FUNCTION_BLOCK AxisHalt IMPLEMENTS I_Task
VAR_INPUT
END_VAR
VAR_OUTPUT
END_VAR
VAR
	mcHalt : Tc2_MC2.MC_Halt;
	_Axis : REFERENCE TO Tc2_MC2.AXIS_REF;
	_Halt : BOOL;
	State: INT;
	_Done: BOOL;
	_Error: BOOL;
	_Busy: BOOL;
END_VAR

{analysis -2}

METHOD Abort : BOOL
mcHalt.Execute := FALSE;
_Busy := FALSE;
_Halt := FALSE;
Abort := TRUE;
State := 0;
END_METHOD

PROPERTY Busy : BOOL
GET
Busy := _Busy;
END_GET
END_PROPERTY

METHOD Cycle : HRESULT
VAR_INPUT
END_VAR
Cycle := S_OK;
CASE State OF
	0:
		IF _Halt THEN
			Cycle := S_PENDING;
			_Done := FALSE;
			_Error := FALSE;
			_Busy := TRUE;
			mcHalt.Execute := TRUE;
			IF mcHalt.Busy THEN
				State := 10;
				_Halt := FALSE;
			END_IF
		END_IF
	
	10:
		IF NOT mcHalt.Busy THEN
			IF mcHalt.Done THEN
				_Done := TRUE;
			ELSIF mcHalt.Error THEN
				_Error := TRUE;
			END_IF
			_Busy := FALSE;
			mcHalt.Execute := FALSE;
			State := 0;
			Cycle := S_OK;
		END_IF
	ELSE
		Cycle := E_FAIL;
END_CASE

mcHalt(Axis := _Axis);
END_METHOD

PROPERTY Deceleration : MC_LREAL
GET
Deceleration := mcHalt.Deceleration;
END_GET
SET
mcHalt.Deceleration := Deceleration;
END_SET
END_PROPERTY

PROPERTY Done : BOOL
GET
Done := _Done;
END_GET
END_PROPERTY

PROPERTY Error : BOOL
GET
Error := _Error;
END_GET
END_PROPERTY

METHOD Execute : HRESULT
VAR_INPUT
	Task : REFERENCE TO I_Task;
END_VAR
IF _Axis.Status.Moving AND NOT _Halt THEN
	Execute := S_OK;
	_Halt := TRUE;
	Task := THIS^;
ELSE
	Execute := S_FALSE;
END_IF
END_METHOD

METHOD FB_init : BOOL
VAR_INPUT
	bInitRetains : BOOL; // if TRUE, the retain variables are initialized (warm start / cold start)
	bInCopyCode : BOOL;  // if TRUE, the instance afterwards gets moved into the copy code (online change)
	axis : reference TO AXIS_REF;
END_VAR
_Axis REF= axis;
END_METHOD

PROPERTY Jerk : MC_LREAL
GET
Jerk := mcHalt.Jerk;
END_GET
SET
mcHalt.Jerk := Jerk;
END_SET
END_PROPERTY

END_FUNCTION_BLOCK

(* stored: Version 1.1.0.1
   POU AxisHalt: Id {8f902aee-94bf-4385-bdcf-ca790f894752}, SpecialFunc None
   Method Abort: Id {628339b1-4bd1-432e-8277-d60f3e75db0d}
   Property Busy: Id {372dcfaa-8cbd-4cb0-a70e-bb4041d8e255}
   Get Get: Id {91d2b55e-e06d-4906-afcd-b4c07ffa30db}
   Method Cycle: Id {82fe1e7b-ab2b-4a89-9b59-5eb25d835959}
   Property Deceleration: Id {268ed3d1-2986-429d-85cd-2c570b60d9d7}
   Get Get: Id {907709a1-b0ba-4945-8711-6554db8f1dc0}
   Set Set: Id {502b45a2-e349-483e-b36a-b0db162a9224}
   Property Done: Id {0d4d59d1-0a33-4a35-91db-70cde82f5006}
   Get Get: Id {5c83bea7-d010-40d8-bc69-060934607785}
   Property Error: Id {3e7959eb-71d7-4ee5-89e9-4dd47b034681}
   Get Get: Id {1eaeb28a-b2d3-41f6-9d16-23d88d0071e2}
   Method Execute: Id {020a5dad-2d55-4c66-8489-dc08945209ce}
   Method FB_init: Id {1d755e0d-6917-492a-87c8-d14e7bb31076}
   Property Jerk: Id {bfb39f13-ace3-4f05-9305-e7d3692f5dfa}
   Get Get: Id {dfdc6efc-8e6e-48e1-a0f4-a06670061327}
   Set Set: Id {9be78a10-cc41-4de6-a2ea-3947cc380f23} *)
